{attribute 'OPC.UA.DA' := '1'}
TYPE Pusher :
STRUCT
	Pusher: BOOL;
	PusherFrontLimit: BOOL;
	PusherBackLimit: BOOL;
END_STRUCT
END_TYPE

(* stored: Version 1.1.0.1, ProductVersion 3.1.4024.12
   DUT Pusher: Id {13e04ccd-6411-484e-bbb0-ee90a32c9016} *)
